FUNCTION_BLOCK PUBLIC ACMethodDosing EXTENDS ACMethodRouteBase
VAR_INPUT
END_VAR
VAR_OUTPUT
END_VAR
VAR PERSISTENT
	_Parameter : ACMethodDosingP;
	_Result : ACMethodDosingR;
END_VAR

PROPERTY IsValid : BOOL
GET
IsValid := TRUE;
END_GET
END_PROPERTY

PROPERTY Parameter : ACMethodDosingP
GET
Parameter := _Parameter;
END_GET
SET // PUBLIC
_Parameter := Parameter;
END_SET
END_PROPERTY

PROPERTY Result : ACMethodDosingR
GET
Result := _Result;
END_GET
SET // PUBLIC
_Result := Result;
END_SET
END_PROPERTY

END_FUNCTION_BLOCK

(* stored: Version 1.1.0.1, ProductVersion 3.1.4022.7
   POU ACMethodDosing: Id {235e2d7a-13fd-4736-b943-188ffb5e542c}, SpecialFunc None
   Property IsValid: Id {c1cdc37e-c84c-45fe-8cf6-fcd5c5bfbf32}
   Get Get: Id {58684e82-97cf-4c8d-acf5-fa08c5d8fb50}
   Property Parameter: Id {fdacd091-5cb1-42e7-8739-78ae4fe6efba}
   Get Get: Id {96313523-9707-4dec-90d8-90b8199f8463}
   Set Set: Id {99fb96e7-ea1a-4b96-8ea5-9d9cf5267075}
   Property Result: Id {357ad5ae-ea13-43fc-b207-8ddbb18c1544}
   Get Get: Id {9a291287-c3c0-4547-a5c8-e4204ddae193}
   Set Set: Id {4ba5b330-4d01-4946-94fe-3881401ee31f} *)
